PROGRAM SAFETY_1


//IF SafetyGlobalVariableList.RUN_STOP = TRUE THEN

//	IF SafetyGlobalVariableList.SAFETY_Permission = FALSE THEN
	
//		CASE SafetyGlobalVariableList.SafetySate OF
		
//			0:
//				SafetyGlobalVariableList.ERR_ACK := FALSE;
//				SafetyGlobalVariableList.SafetySate := SafetyGlobalVariableList.SafetySate + 10;
//			10:
//				SafetyGlobalVariableList.ERR_ACK := TRUE;
//				SafetyGlobalVariableList.SafetySate := SafetyGlobalVariableList.SafetySate + 10;
//			20:
//				SafetyGlobalVariableList.ERR_ACK := FALSE;
//				SafetyGlobalVariableList.SafetySate := SafetyGlobalVariableList.SafetySate + 10;
//			30:		
//				SafetyGlobalVariableList.AX5805_ErrACK := FALSE;
//				SafetyGlobalVariableList.SafetySate := SafetyGlobalVariableList.SafetySate + 10;
//			40:	
//				SafetyGlobalVariableList.AX5805_ErrACK := TRUE;
//				SafetyGlobalVariableList.SafetySate := SafetyGlobalVariableList.SafetySate + 10;
//			50:
//				SafetyGlobalVariableList.AX5805_ErrACK := FALSE;
//				SafetyGlobalVariableList.SafetySate := SafetyGlobalVariableList.SafetySate + 10;	
//			60:
//				SafetyGlobalVariableList.RestartFBs_TSG := FALSE;
//				SafetyGlobalVariableList.SafetySate := SafetyGlobalVariableList.SafetySate + 10;
//			70:
//				SafetyGlobalVariableList.RestartFBs_TSG := TRUE;
//				SafetyGlobalVariableList.SafetySate := SafetyGlobalVariableList.SafetySate + 10;	
//			80:
//				SafetyGlobalVariableList.RestartFBs_TSG := FALSE;
//				SafetyGlobalVariableList.SafetySate := SafetyGlobalVariableList.SafetySate + 10;	
//			90:		
//				SafetyGlobalVariableList.SafetySate := 0;

//		END_CASE
//	END_IF	

//END_IF

END_PROGRAM

(* stored: Version 1.1.0.1, ProductVersion 3.1.4024.15
   POU SAFETY_1: Id {fe3eb017-1e4d-407b-90fe-7196ffdfbcaf}, SpecialFunc None *)
